// TwinCAT 3 PLC project igen
// ProgramVersion: 3.1.4024.0
// libraries:
//   Tc2_Standard, * (Beckhoff Automation GmbH)
//   Tc2_System, * (Beckhoff Automation GmbH)
//   Tc3_Module, * (Beckhoff Automation GmbH)
// project tree:
//   GVLs/ GVL_1.TcGVL
//   / PlcTask.TcTTO
//   POUs/ CallHandler.TcPOU, DoorControl.TcPOU, DoorSensors.TcPOU, Lights.TcPOU, MAIN.TcPOU, MovementControl.TcPOU, TargetFloorLights.TcPOU

CONFIGURATION igen
    RESOURCE PLC ON TwinCAT3
        TASK PlcTask(INTERVAL := T#10ms, PRIORITY := 20);
        PROGRAM MAIN WITH PlcTask : MAIN;
    END_RESOURCE
END_CONFIGURATION

// ---- GVLs/GVL_1.TcGVL
VAR_GLOBAL
    i_bCallButtons : ARRAY[0..10] OF BOOL;
    i_bCallUp : ARRAY[1..9] OF BOOL;
    i_bCallDown : ARRAY[1..9] OF BOOL;
    i_bDoorClosed : BOOL;
    i_bDoorOpen : BOOL;
    i_iCurrentFloor : INT;

    q_bMoveUp AT %Q* : BOOL;
    q_bMoveDown AT %Q* : BOOL;
    q_bOpenDoor AT %Q* : BOOL;
    q_bCloseDoor AT %Q* : BOOL;
    q_bCallAckUp AT %Q* : ARRAY[1..9] OF BOOL;
    q_bCallAckDown AT %Q* : ARRAY[1..9] OF BOOL;

    g_iTargetFloor : INT;
    g_bDoorTimerActive : BOOL;
    g_bCallRegisteredUp : ARRAY[1..9] OF BOOL;
    g_bCallRegisteredDown : ARRAY[1..9] OF BOOL;
    g_bMovingUp : BOOL;
    g_bMovingDown : BOOL;
END_VAR

// ---- POUs/MAIN.TcPOU
PROGRAM MAIN
VAR
    fb_CallHandler : CallHandler;
    fb_MovementControl : MovementControl;
    fb_DoorControl : DoorControl;
	fb_DoorSensors : DoorSensors;
	fb_Lights : Lights;
	fb_TargetFloorLights : TargetFloorLights;
END_VAR

fb_CallHandler();
fb_DoorControl();
fb_MovementControl();
fb_DoorSensors();
fb_Lights();
fb_TargetFloorLights();

END_PROGRAM

// ---- POUs/CallHandler.TcPOU
FUNCTION_BLOCK CallHandler
VAR_INPUT
END_VAR
VAR_OUTPUT
END_VAR
VAR
	r_i: INT;
	doorOpenTimer : TON;
END_VAR

FOR r_i := 0 TO 10 DO
    IF GVL_1.i_bCallButtons[r_i] THEN
        GVL_1.g_iTargetFloor := r_i;
        RETURN;
    END_IF;
END_FOR

IF GVL_1.g_bMovingUp THEN
    FOR r_i := GVL_1.i_iCurrentFloor + 1 TO 9 DO
        IF GVL_1.i_bCallUp[r_i] THEN
            GVL_1.g_iTargetFloor := r_i;
            RETURN;
        END_IF;
    END_FOR
END_IF

IF GVL_1.g_bMovingDown THEN
    r_i := GVL_1.i_iCurrentFloor - 1;
    WHILE r_i >= 1 DO
        IF GVL_1.i_bCallDown[r_i] THEN
            GVL_1.g_iTargetFloor := r_i;
            RETURN;
        END_IF;
        r_i := r_i - 1;
    END_WHILE;
END_IF

IF NOT GVL_1.g_bMovingUp AND NOT GVL_1.g_bMovingDown THEN
    FOR r_i := 1 TO 9 DO
        IF GVL_1.i_bCallUp[r_i] OR GVL_1.i_bCallDown[r_i] THEN
            GVL_1.g_iTargetFloor := r_i;
            RETURN;
        END_IF;
    END_FOR
END_IF

IF GVL_1.i_iCurrentFloor = GVL_1.g_iTargetFloor THEN
    GVL_1.q_bOpenDoor := TRUE;
    doorOpenTimer(IN := TRUE, PT := T#10S);
    IF doorOpenTimer.Q THEN
        GVL_1.q_bOpenDoor := FALSE;
        GVL_1.q_bCloseDoor := TRUE;
        doorOpenTimer(IN := FALSE);

        GVL_1.i_bCallUp[GVL_1.g_iTargetFloor] := FALSE;
        GVL_1.i_bCallDown[GVL_1.g_iTargetFloor] := FALSE;
    END_IF
ELSE
    doorOpenTimer(IN := FALSE);
END_IF

END_FUNCTION_BLOCK

// ---- POUs/MovementControl.TcPOU
FUNCTION_BLOCK MovementControl
VAR_INPUT
END_VAR
VAR_OUTPUT
END_VAR
VAR
	r_reachedTarget : BOOL;
	r_timer : TON;
END_VAR

r_reachedTarget := (GVL_1.i_iCurrentFloor = GVL_1.g_iTargetFloor);

IF GVL_1.i_bDoorClosed THEN
    IF NOT r_reachedTarget THEN
        IF GVL_1.i_iCurrentFloor < GVL_1.g_iTargetFloor THEN
            GVL_1.q_bMoveUp := TRUE;
            GVL_1.q_bMoveDown := FALSE;
            GVL_1.i_iCurrentFloor := GVL_1.i_iCurrentFloor + 1;
        END_IF

        IF GVL_1.i_iCurrentFloor > GVL_1.g_iTargetFloor THEN
            GVL_1.q_bMoveUp := FALSE;
            GVL_1.q_bMoveDown := TRUE;
            GVL_1.i_iCurrentFloor := GVL_1.i_iCurrentFloor - 1;
        END_IF
    ELSE
        GVL_1.q_bMoveUp := FALSE;
        GVL_1.q_bMoveDown := FALSE;
    END_IF
END_IF

END_FUNCTION_BLOCK

// ---- POUs/DoorControl.TcPOU
FUNCTION_BLOCK DoorControl
VAR_INPUT
END_VAR
VAR_OUTPUT
END_VAR
VAR
	r_doorTimer : TON;
END_VAR

//GVL_1.q_bOpenDoor := FALSE;
//GVL_1.q_bCloseDoor := FALSE;

IF GVL_1.i_iCurrentFloor = GVL_1.g_iTargetFloor THEN
    GVL_1.q_bOpenDoor := TRUE;
	GVL_1.q_bCloseDoor := FALSE;
    r_doorTimer(IN := TRUE, PT := T#10S);
ELSE
    GVL_1.q_bCloseDoor := TRUE;
	GVL_1.q_bOpenDoor := FALSE;
    r_doorTimer(IN := FALSE);
END_IF

IF r_doorTimer.Q THEN
    GVL_1.q_bOpenDoor := FALSE;
    GVL_1.q_bCloseDoor := TRUE;
	r_doorTimer(IN := FALSE);
END_IF

END_FUNCTION_BLOCK

// ---- POUs/DoorSensors.TcPOU
FUNCTION_BLOCK DoorSensors
VAR_INPUT
END_VAR
VAR_OUTPUT
END_VAR
VAR
	r_doorCloseTimer : TON;
	r_doorOpenError : BOOL;
END_VAR

r_doorOpenError := FALSE;

IF NOT GVL_1.i_bDoorClosed THEN
    r_doorCloseTimer(IN := TRUE, PT := T#5S);
    
    IF r_doorCloseTimer.Q THEN
        r_doorOpenError := TRUE;
		r_doorCloseTimer(IN := FALSE);
    END_IF
ELSE
    r_doorCloseTimer(IN := FALSE);
    r_doorOpenError := FALSE;
END_IF
IF r_doorOpenError THEN
    GVL_1.q_bMoveUp := FALSE;
    GVL_1.q_bMoveDown := FALSE;
END_IF

END_FUNCTION_BLOCK

// ---- POUs/Lights.TcPOU
FUNCTION_BLOCK Lights
VAR_INPUT
END_VAR
VAR_OUTPUT
END_VAR
VAR
	r_i: INT;
END_VAR

FOR r_i := 1 TO 9 DO
    IF GVL_1.i_bCallUp[r_i] THEN
        GVL_1.q_bCallAckUp[r_i] := TRUE;
    END_IF
    
    IF GVL_1.i_bCallDown[r_i] THEN
        GVL_1.q_bCallAckDown[r_i] := TRUE;
    END_IF

    IF GVL_1.i_iCurrentFloor = r_i AND GVL_1.i_bDoorOpen AND 
       (GVL_1.q_bCallAckUp[r_i] OR GVL_1.q_bCallAckDown[r_i]) THEN
        GVL_1.q_bCallAckUp[r_i] := FALSE;
        GVL_1.q_bCallAckDown[r_i] := FALSE;
        GVL_1.i_bCallUp[r_i] := FALSE;
        GVL_1.i_bCallDown[r_i] := FALSE;
    END_IF
END_FOR

FOR r_i := 0 TO 10 DO
    IF GVL_1.i_bCallButtons[r_i] AND GVL_1.i_iCurrentFloor = r_i THEN
        GVL_1.q_bOpenDoor := TRUE;
    END_IF
END_FOR

END_FUNCTION_BLOCK

// ---- POUs/TargetFloorLights.TcPOU
FUNCTION_BLOCK TargetFloorLights
VAR_INPUT
END_VAR
VAR_OUTPUT
END_VAR
VAR
	r_i: INT;
END_VAR

FOR r_i := 0 TO 10 DO
	IF GVL_1.i_bCallButtons[r_i] THEN
		GVL_1.q_bOpenDoor := TRUE;
	END_IF
END_FOR

END_FUNCTION_BLOCK
